Fanuc KAREL source: CA0046.KL

PROGRAM CA0046
%STACKSIZE=65535
%PRIORITY=65535
%NOLOCKGROUP
VAR
G : INTEGER
I : INTEGER
R : REAL
B : BOOLEAN
S : STRING[16]
AI : ARRAY[2] OF INTEGER
AR : ARRAY[2] OF REAL
P : XYZWPR
-- UNRESOLVED DECLARATIONS (source type spelling not recovered)
-- ST : TYPE_0x1100 (type_u16=0x1100)
-- V : TYPE_0x0013 (type_u16=0x0013)
ROUTINE F(P1 : ARRAY[*] OF INTEGER; P2 : ARRAY[*] OF REAL; P3 : TYPE_0x1100; P4 : XYZWPR; P5 : TYPE_0x0013; P6 : ARRAY[*] OF INTEGER; P7 : ARRAY[*] OF REAL; P8 : TYPE_0x1100; P9 : XYZWPR; P10 : TYPE_0x0013; P11 : ARRAY[*] OF INTEGER;
P12 : ARRAY[*] OF REAL; P13 : TYPE_0x1100; P14 : XYZWPR; P15 : TYPE_0x0013; P16 : ARRAY[*] OF INTEGER; P17 : ARRAY[*] OF REAL; P18 : TYPE_0x1100; P19 : XYZWPR; P20 : TYPE_0x0013; P21 : ARRAY[*] OF INTEGER;
P22 : ARRAY[*] OF REAL; P23 : TYPE_0x1100; P24 : XYZWPR) FROM CA0046
ROUTINE F
BEGIN
G=(G + 1)
END F
BEGIN
G=0
I=1
R=2.5
B=TRUE
S='A'
AI[1]=3
AR[1]=4.5
ST.A=5
ST.B=1087373312
F(AI,AR,ST,P,V,AI,AR,ST,P,V,AI,AR,ST,P,V,AI,AR,ST,P,V,AI,AR,ST,P)
END CA0046
